// TIA Portal V19 export
DATA_BLOCK "Com_ToFruitPlantAlsafe"   // DB305
{ S7_Optimized_Access := 'TRUE' }
// stored: AutoNumber false, MemoryReserve 0
   VAR RETAIN
      AFM1 : Struct   // Signals From Ampack
         Ready : Bool;   // Ready for production
         Prod_Fruit_Req : Bool;   // Request Fruit product
         Filler1_ProductPumpReq : Bool;   // Product Pump Request
         Ready_For_CIP : Bool;   // Ready for CIP - Not Used
         GS22_61 : Bool;   // APV AHV- FP1 - Route to Polygon Filler - Flow Bend Connected
         GS22_62 : Bool;   // APV AHV- FP1 - Route to Polygon Filler - Blank Fitted
         CIP_Prod_Clusters : Bool;   // Information - Product clusters cleaning - Use to interlock sterilisation
         PG_TransferLine_Clean : Bool;   // Gemini HMI indication
         PG_TransferLine_Sterile : Bool;   // Gemini HMI indication
         SpareBool_1_1 : Bool;
         SpareBool_1_2 : Bool;
         SteamBarrierActv_PD_CL2 : Bool;   // Steam barrier activated pre doser product cluster 2 - Fruit
         SpareBool_1_4 : Bool;
         SpareBool_1_5 : Bool;
         SpareBool_1_6 : Bool;
         SpareBool_1_7 : Bool;
         SpareBool_2_0 : Bool;
         SpareBool_2_1 : Bool;
         SpareBool_2_2 : Bool;
         SpareBool_2_3 : Bool;
         SpareBool_2_4 : Bool;
         SpareBool_2_5 : Bool;
         SpareBool_2_6 : Bool;
         SpareBool_2_7 : Bool;
         SpareBool_3_0 : Bool;
         SpareBool_3_1 : Bool;
         SpareBool_3_2 : Bool;
         SpareBool_3_3 : Bool;
         SpareBool_3_4 : Bool;
         SpareBool_3_5 : Bool;
         SpareBool_3_6 : Bool;
         SpareBool_3_7 : Bool;
         SpareBool_4_0 : Bool;
         SpareBool_4_1 : Bool;
         SpareBool_4_2 : Bool;
         SpareBool_4_3 : Bool;
         SpareBool_4_4 : Bool;
         SpareBool_4_5 : Bool;
         SpareBool_4_6 : Bool;
         SpareBool_4_7 : Bool;
         Nom_FillgLev_PD : Int;   // Not used
         Nom_FillgLev_MD1 : Int;   // Not used
         Nom_FillgLev_MD2 : Int;   // Not used
         Actl_FillgLev_PD : Int;   // Not used
         Actl_FillgLev_MD1 : Int;   // Not used
         Actl_FillgLev_MD2 : Int;   // Not used
         REM_WD_CNT : Int;
      END_STRUCT;
      hmi : Struct
         commsFault : Bool;
         s1 : Bool;   // spare
         s2 : Bool;   // spare
         s3 : Bool;   // spare
         s4 : Bool;   // spare
         s5 : Bool;   // spare
         s6 : Bool;   // spare
         s7 : Bool;   // spare
         s8 : Bool;   // spare
         s9 : Bool;   // spare
         s10 : Bool;   // spare
         s11 : Bool;   // spare
         s12 : Bool;   // spare
         s13 : Bool;   // spare
         s14 : Bool;   // spare
         s15 : Bool;   // spare
      END_STRUCT;
      Spare : Array[0..36] of Byte;
   END_VAR
BEGIN
END_DATA_BLOCK
